FUNCTION_BLOCK FB_Machine EXTENDS FB_Module
VAR_INPUT
END_VAR
VAR_OUTPUT
END_VAR
VAR
	fbEthercatDiagnostic:	FB_EthercatDiagnostic<10>;
END_VAR

// https://peterzerlauth.com/

fbEthercatDiagnostic();

SUPER^();

METHOD PROTECTED M_Execute : BOOL
VAR_INPUT
END_VAR
VAR
	bReturn:					BOOL:= TRUE;
END_VAR
M_Execute:= TRUE;
END_METHOD

METHOD PROTECTED M_Starting : BOOL
VAR_INPUT
END_VAR
M_Starting:= SUPER^.M_Starting();
END_METHOD

METHOD PROTECTED M_Stopping : BOOL // Return state complete
VAR_INPUT
END_VAR
// State Stopping
M_Stopping:= SUPER^.M_Stopping();
END_METHOD

END_FUNCTION_BLOCK

(* stored: Version 1.1.0.1
   POU FB_Machine: Id {3de86606-a9be-0cdd-161e-36bed1c57924}, SpecialFunc None
   Method M_Execute: Id {45dd9f3e-d6f6-04de-33c0-4769c77fb584}
   Method M_Starting: Id {285faf55-e10d-03d6-26f0-866c85f1872d}
   Method M_Stopping: Id {d97ed520-4549-0067-3e89-5d2dbde992b2} *)
